KUKA KRL program: hp040.src, hp040.dat

--- hp040.src ---
&ACCESS RVP
&REL 5
&COMMENT Axor LTA
&PARAM TEMPLATE = C:\KRC\ROBOTER\TEMPLATE\VG_HP
&PARAM EDITMASK = *
DEF hp040( )
EXT CHECK_RIGHT_TOOL()
;FOLD INI;%{PE}%V3.2.0,%MKUKATPBASIS,%CINIT,%VCOMMON,%P
;FOLD BAS INI;%{E}%V3.2.0,%MKUKATPBASIS,%CINIT,%VINIT,%P
    GLOBAL INTERRUPT DECL 3 WHEN $STOPMESS==TRUE DO IR_STOPM ( )
    INTERRUPT ON 3
    BAS (#INITMOV,0)
;ENDFOLD (BAS INI)
;FOLD GRIPPER INI;%{E}%V3.2.0,%MKUKATPGRIPPER,%CINIT,%VINIT,%P
    USER_GRP(0,DUMMY,DUMMY,GDEFAULT)
;ENDFOLD (GRIPPER INI)
;FOLD SPOT INI;%{E}%V3.2.0,%MKUKATPSPOT,%CINIT,%VINIT,%P
    USERSPOT(#INIT)
;ENDFOLD (SPOT INI)
;FOLD USER INI;%{E}%V3.2.0,%MKUKATPUSER,%CINIT,%VINIT,%P
;Make your modifications here
;FOLD COLLISION_V_3.01 INI ;%{E}
    IF (COLLISION_DATA[1].I_NR>0) THEN
         GLOBAL INTERRUPT DECL 21 WHEN $IN[COLLISION_DATA[1].I_NR]==FALSE DO COLLSTOP (1,0 )
    ENDIF
    IF (COLLISION_DATA[2].I_NR>0) THEN
         GLOBAL INTERRUPT DECL 22 WHEN $IN[COLLISION_DATA[2].I_NR]==FALSE DO COLLSTOP (2,0 )
    ENDIF
    IF (COLLISION_DATA[3].I_NR>0) THEN
         GLOBAL INTERRUPT DECL 23 WHEN $IN[COLLISION_DATA[3].I_NR]==FALSE DO COLLSTOP (3,0 )
    ENDIF
    IF (COLLISION_DATA[4].I_NR>0) THEN
         GLOBAL INTERRUPT DECL 24 WHEN $IN[COLLISION_DATA[4].I_NR]==FALSE DO COLLSTOP (4,0 )
    ENDIF
;ENDFOLD
;ENDFOLD (USER INI)
;ENDFOLD (INI)

; Caracterizacao dos meios de producao
; Changes: HP040 - Axor LTA
; Versao Atual: 27/03/2016
; Name: P13.060-R3

$TIMER[1]=0
$TIMER_STOP[1]=FALSE

chk_w1_wechs_ok ( )        ; CHECK GUN C1

MBINI( )                   ; RESET SINAIS

;FOLD PTP HOME  Vel= 100 % DEFAULT;%{PE}%V3.2.0,%MKUKATPBASIS,%CMOVE,%VPTP,%P 1:PTP, 2:HOME, 3:, 5:100, 7:DEFAULT
$BWDSTART = FALSE
$H_POS=XHOME
PDAT_ACT=PDEFAULT
BAS(#PTP_DAT)
FDAT_ACT=FHOME
BAS(#FRAMES)
BAS(#VEL_PTP,100)
PTP XHOME
;ENDFOLD

ps_b_lta_res_c01 ( )       ; SOLDA RESPOT C1

WKZ1_AB ( )                ; DEPOSITA PINCA C1

WKZ4_AN ( )                ; PEGA PINCA C2

ps_b_lta_res_c02 ( )       ; SOLDA RESPOT C2

WKZ4_AB ( )                ; DEPOSITA PINCA C2

perfil_livre ( )           ; PERFIL LIVRE ESTACAO

trabalho_concluido ( )     ; TRABALHO CONCLUIDO

WKZ1_AN ( )                ; PEGA PINCA C1

;FOLD PTP HOME  Vel= 100 % DEFAULT;%{PE}%V3.2.0,%MKUKATPBASIS,%CMOVE,%VPTP,%P 1:PTP, 2:HOME, 3:, 5:100, 7:DEFAULT
$BWDSTART = FALSE
$H_POS=XHOME
PDAT_ACT=PDEFAULT
BAS(#PTP_DAT)
FDAT_ACT=FHOME
BAS(#FRAMES)
BAS(#VEL_PTP,100)
PTP XHOME
;ENDFOLD

$TIMER_STOP[1]=TRUE

END

--- hp040.dat ---
&ACCESS RVP
&REL 5
&COMMENT Axor LTA
&PARAM TEMPLATE = C:\KRC\ROBOTER\TEMPLATE\VG_HP
&PARAM EDITMASK = *
DEFDAT hp040
;FOLD EXTERNAL DECLARATIONS;%{PE}%V2.2.2,%MKUKATPBASIS,%CEXT,%VCOMMON,%P
;FOLD BAS EXT;%{PE}%V2.2.2,%MKUKATPBASIS,%CEXT,%VEXT,%P
EXT  BAS (BAS_COMMAND  :IN,REAL  :IN )
DECL INT SUCCESS
;ENDFOLD
;FOLD A10 EXT;%{E}%V2.2.2,%MKUKATPARC,%CEXT,%VEXT,%P
EXT  A10 (A_CMD_T  :IN,A_STRT_T  :IN,A_WELD_T  :IN,A_END_T  :IN,INT  :IN )
;ENDFOLD
;FOLD A20 EXT;%{E}%V2.2.2,%MKUKATPA20,%CEXT,%VEXT,%P
EXT  A20 (INT  :IN,WELD_ST  :IN,WELD_FI  :IN,INT  :IN )
;ENDFOLD
;FOLD GRIPPER EXT;%{E}%V2.2.2,%MKUKATPGRIPPER,%CEXT,%VEXT,%P
EXT  H50 (INT  :IN,INT  :IN,INT  :IN,GRP_TYP  :IN )
;ENDFOLD
;FOLD SPOT EXT;%{E}%V2.2.2,%MKUKATPSPOT,%CEXT,%VEXT,%P
EXT  USERSPOT (S_COMMAND  :IN,SPOT_TYPE  :IN )
;ENDFOLD
;FOLD TOUCHSENSE EXT;%{E}%V2.2.2,%MKUKATPTS,%CEXT,%VEXT,%P
EXT  H70 (INT  :IN,SRCH_TYP_2  :OUT,E6POS  :IN,SRCH_TYP_3  :IN,SRCH_TYP_2  :IN,SRCH_TYP_2  :IN,SRCH_TYP_2  :IN,SRCH_TYP_2  :IN,SRCH_TYP_2  :IN,INT  :IN )
;ENDFOLD
;FOLD USER EXT;%{}%V2.2.2,%MKUKATPUSER,%CEXT,%VEXT,%P
;Make here your modifications
;ENDFOLD
;ENDFOLD

ENDDAT
